FUNCTION_BLOCK CM_AX5000 EXTENDS CM_Base IMPLEMENTS I_AX5000
VAR_INPUT
	i_refAxis : REFERENCE TO Tc2_MC2.AXIS_REF;
	i_bIclkForward : BOOL := TRUE; //TRUE = interlocked
	i_bIclkBackward : BOOL := TRUE; //TRUE = interlocked
END_VAR

VAR
	fbPower : Tc2_MC2.MC_Power;
	fbReset : Tc2_MC2.MC_Reset;
	fbHome : Tc2_MC2.MC_Home;
	fbJog : Tc2_MC2.MC_Jog;
	fbMoveAbsolute : Tc2_MC2.MC_MoveAbsolute;
	fbMoveRelative : Tc2_MC2.MC_MoveRelative;
	fbStop : Tc2_MC2.MC_Stop;	

	// Inputs
	I_bDetReferenceSwitch AT %I* : BOOL; //Reference-/home switch
	I_bDetLimitSwitchPositive AT %I* : BOOL; //Limit switch positive-/CW- direction
	I_bDetLimitSwitchNegative AT %I* : BOOL; //Limit switch negative-/CCW- direction
	
	//Properties
	s_bStatus : BOOL;
	s_bDone : BOOL; 
	s_bBusy : BOOL; 
	s_bActive : BOOL; 
	s_bCommandAborted : BOOL; 
	s_bError : BOOL; 
	s_nErrorID : UDINT;
	
	// Requests
	{warning '#TODO: Chcek / update during develiping'}
	s_bReqStop : BOOL;
	s_bReqStartForward : BOOL;
	s_bReqStartBackward : BOOL;
	s_bReqReset : BOOL;
	
	// Commands
	s_bCmdEnable : BOOL;
	s_bCmdReset : BOOL;
	s_bCmdForward : BOOL;
	s_bCmdBackward : BOOL;
	s_bCmdReleaseBrake : BOOL;
		
	// States
	s_bStaReadyForOperation: BOOL;
	s_bStaDriveError: BOOL;
	s_bStaWarning : BOOL;
	
	
	
	s_sInterlockedReason : STRING; //External interlocked reason for clarifying reason
	
	// Setpoints
	s_fTargetSpeed : LREAL; // Target speed [mm/s]
	
	// Timers
	
	// Alarms
	s_fbAlarmHandlerDriveError : FB_AlarmHandler;
	s_fbAlarmHandlerStartMotorNotAllowed : FB_AlarmHandler;
	s_fbAlarmHandlerMotorForwardInterlocked : FB_AlarmHandler;
	s_fbAlarmHandlerMotorBackwardInterlocked : FB_AlarmHandler;
	
	s_errDriveError : BOOL;
	s_wrnStartMotorNotAllowed : BOOL;
	s_wrnMotorForwardInterlocked : BOOL;
	s_wrnMotorBackwardInterlocked : BOOL;
	
	//Hmi
	s_fbHmiBtnManualForward		: FB_HmiBtn;
	s_fbHmiBtnManualBackward	: FB_HmiBtn;
	s_fbHmiBtnManualStop		: FB_HmiBtn;
	s_fbHmiBtnManualReset		: FB_HmiBtn;
	
	s_fbHmiLedMotorStopped		: FB_HmiLed;
	s_fbHmiLedDriveError		: FB_HmiLed;
	
	//Sequence
	eSeqMOVITRAC_B_WithBrake : E_SeqMOVITRAC_B_WithBrake;
	seqTimer : TON;
	seqPreStep : E_SeqMOVITRAC_B_WithBrake;
	s_sActStep : STRING;
	
END_VAR


SUPER^();

METHOD PUBLIC m_MC_Home : BOOL
VAR_INPUT
	i_bExecute : BOOL;
	i_fPosition : REAL;
	i_eHomingMode : TC2_MC2.MC_HomingMode;
	i_eBufferMode : TC2_MC2.MC_BufferMode;
END_VAR

fbHome(
	Axis := i_refAxis,
	Execute := i_bExecute,
	Position := i_fPosition,
	HomingMode := i_eHomingMode,
	BufferMode := i_eBufferMode,
	Options := ,
	bCalibrationCam := I_bDetReferenceSwitch,
	Done => s_bDone,
	Busy => s_bBusy,
	Active => s_bActive,
	CommandAborted => s_bCommandAborted,
	Error => s_bError,
	ErrorID => s_nErrorID);
	
m_MC_Home := s_bDone;
END_METHOD

METHOD PUBLIC m_MC_Jog : BOOL
VAR_INPUT
	i_bExecute : BOOL;
	i_bJogForward : BOOL;
	i_bJogBackward : BOOL;
	i_eJogMode : TC2_MC2.E_JogMode;
	i_fPosition : LREAL; 
	i_fVelocity : LREAL; 
	i_fAcceleration : LREAL; 
	i_fDeceleration : LREAL; 
	i_fJerk : LREAL;
END_VAR

fbJog(
	Axis := i_refAxis,
	JogForward := i_bJogForward,
	JogBackwards := i_bJogBackward,
	Mode := i_eJogMode,
	Position := i_fPosition,
	Velocity := i_fVelocity,
	Acceleration := i_fAcceleration,
	Deceleration := i_fDeceleration,
	Jerk := i_fJerk,
	Done => s_bDone,
	Busy => s_bBusy,
	Active => s_bActive,
	CommandAborted => s_bCommandAborted,
	Error => s_bError,
	ErrorID => s_nErrorID);
	
m_MC_Home := s_bDone;
END_METHOD

METHOD PUBLIC m_MC_MoveAbsolute : BOOL
VAR_INPUT
	i_bExecute : BOOL;
	i_fPosition : LREAL; 
	i_fVelocity : LREAL; 
	i_fAcceleration : LREAL; 
	i_fDeceleration : LREAL; 
	i_fJerk : LREAL;
	i_eBufferMode : TC2_MC2.MC_BufferMode;
END_VAR

fbMoveAbsolute(
	Axis := i_refAxis,
	Execute := i_bExecute, 
	Position := i_fPosition,
	Velocity := i_fVelocity,
	Acceleration := i_fAcceleration,
	Deceleration := i_fDeceleration,
	Jerk := i_fJerk,
	BufferMode := i_eBufferMode,
	Options := ,
	Done => s_bDone,
	Busy => s_bBusy,
	Active => s_bActive,
	CommandAborted => s_bCommandAborted,
	Error => s_bError,
	ErrorID => s_nErrorID);
	
m_MC_Home := s_bDone;
END_METHOD

METHOD PUBLIC m_MC_MoveRelative : BOOL
VAR_INPUT
	i_bExecute : BOOL;
	i_fDistance : LREAL; 
	i_fVelocity : LREAL; 
	i_fAcceleration : LREAL; 
	i_fDeceleration : LREAL; 
	i_fJerk : LREAL;
	i_eBufferMode : TC2_MC2.MC_BufferMode;
END_VAR

fbMoveRelative(
	Axis := i_refAxis,
	Execute := i_bExecute,
	Distance := i_fDistance,
	Velocity := i_fVelocity,
	Acceleration := i_fAcceleration,
	Deceleration := i_fDeceleration,
	Jerk := i_fJerk,
	BufferMode := i_eBufferMode,
	Options := ,
	Done => s_bDone,
	Busy => s_bBusy,
	Active => s_bActive,
	CommandAborted => s_bCommandAborted,
	Error => s_bError,
	ErrorID => s_nErrorID);
	
m_MC_Home := s_bDone;
END_METHOD

METHOD PUBLIC m_MC_Power : BOOL
VAR_INPUT
	i_bEnable : BOOL;
	i_bEnablePositive : BOOL;
	i_bEnableNegative : BOOL;
	i_fOverride : LREAL;
	i_eBufferMode : TC2_MC2.MC_BufferMode;
END_VAR

fbPower(
	Axis := i_refAxis,
	Enable := i_bEnable,
	Enable_Positive := i_bEnablePositive,
	Enable_Negative := i_bEnableNegative,
	Override := i_fOverride,
	BufferMode := i_eBufferMode,
	Options := ,
	Status => s_bStatus,
	Busy => s_bBusy,
	Active => s_bActive,
	Error => s_bError,
	ErrorID => s_nErrorID);

m_MC_Home := s_bDone;
END_METHOD

METHOD PUBLIC m_MC_Reset : BOOL
VAR_INPUT
	i_bExecute : BOOL;
END_VAR

fbReset(
	Axis := i_refAxis,
	Execute := i_bExecute,
	Done => s_bDone,
	Busy => s_bBusy,
	Error => s_bError,
	ErrorID => s_nErrorID);

m_MC_Home := s_bDone;
END_METHOD

METHOD PUBLIC m_MC_Stop : BOOL
VAR_INPUT
	i_bExecute : BOOL;
	i_fDeceleration : LREAL;
	i_fJerk : LREAL;
END_VAR

fbStop(
	Axis := i_refAxis,
	Execute := i_bExecute,
	Deceleration := i_fDeceleration,
	Jerk := i_fJerk,
	Options := ,
	Done => s_bDone,
	Busy => s_bBusy,
	Active => s_bActive,
	CommandAborted => s_bCommandAborted,
	Error => s_bError,
	ErrorID => s_nErrorID);


m_MC_Home := s_bDone;
END_METHOD

PROPERTY PUBLIC p_bActive : BOOL
GET

p_bActive := s_bActive;
END_GET
END_PROPERTY

PROPERTY PUBLIC p_bBusy : BOOL
GET

p_bBusy := s_bBusy;
END_GET
END_PROPERTY

PROPERTY PUBLIC p_bCommandAborted : BOOL
GET

p_bCommandAborted := s_bCommandAborted
END_GET
END_PROPERTY

PROPERTY PUBLIC p_bDone : BOOL
GET

p_bDone := s_bDone
END_GET
END_PROPERTY

PROPERTY PUBLIC p_bError : BOOL
GET

p_bError := s_bError;
END_GET
END_PROPERTY

PROPERTY PUBLIC p_bHomed : BOOL
GET

p_bHomed := i_refAxis.Status.Homed;
END_GET
END_PROPERTY

PROPERTY PUBLIC p_bStandstill : BOOL
GET

p_bStandstill := i_refAxis.Status.StandStill;
END_GET
END_PROPERTY

PROPERTY PUBLIC p_fPosition : LREAL
GET

p_fPosition := i_refAxis.NcToPlc.ActPos;
END_GET
END_PROPERTY

PROPERTY PUBLIC p_fVelocity : LREAL
GET

p_fVelocity := i_refAxis.NcToPlc.ActVelo;
END_GET
END_PROPERTY

PROPERTY PUBLIC p_nErrorID : UDINT
GET

p_nErrorID := s_nErrorID;
END_GET
END_PROPERTY

END_FUNCTION_BLOCK

(* stored: Version 1.1.0.1, ProductVersion 3.1.4024.12
   POU CM_AX5000: Id {29dfdbae-f16d-497a-b262-2baea4701d77}, SpecialFunc None
   Folder Methods: Id {c7dc02dc-f2cb-44e5-89eb-2e4085b6a909}
   Folder Properties: Id {c3e008a7-9dfe-49e0-9cc5-18c79327535a}
   Method m_MC_Home: Id {953753d2-b56b-4416-8bfe-ffc202c2c66e}
   Method m_MC_Jog: Id {0b34f7cb-ad06-475a-9339-58c1a8e417e5}
   Method m_MC_MoveAbsolute: Id {0f6a7ef6-bbb9-453d-8d82-3eac920331b1}
   Method m_MC_MoveRelative: Id {e88d3f53-895e-4d90-93a1-00c818a65e17}
   Method m_MC_Power: Id {fd1fc676-b701-4a26-938f-ef477da725d4}
   Method m_MC_Reset: Id {78a60c41-19c8-4eb1-aa13-d3edbd9b9522}
   Method m_MC_Stop: Id {6c6294b9-0bc1-4c87-8f3e-41d07e1a757c}
   Property p_bActive: Id {fdebd466-4355-4961-86f7-17cb1e74e332}
   Get Get: Id {12554b68-dea8-473b-b98f-bf82edb9ad16}
   Property p_bBusy: Id {a6bb4214-9e42-46dd-a8f3-995e364772d0}
   Get Get: Id {7080bc48-c94e-419b-9e7d-df95694c753e}
   Property p_bCommandAborted: Id {32bd9d7d-f5a3-4f89-9a59-0294a826c560}
   Get Get: Id {a39acfdd-fde9-4118-9e65-bd86ad5a94af}
   Property p_bDone: Id {09a3960b-0e70-4e33-a3d6-ff5a57122d42}
   Get Get: Id {e656286c-fa2b-43ef-a794-1f2819d97be9}
   Property p_bError: Id {7759aec3-bd8b-4f0c-9913-656b2c70cf6a}
   Get Get: Id {67b5f8fe-c6e4-4145-9f0e-f9d36c480d63}
   Property p_bHomed: Id {29d86fc1-be45-4333-91ce-9bdc79739fba}
   Get Get: Id {3bff5f71-c84f-4863-9be2-8ae02d95a4db}
   Property p_bStandstill: Id {06fe4adf-3a6b-49c2-a8e8-c5de29d0c1af}
   Get Get: Id {e4db3dbb-9fbf-4ca7-ba91-332924a328ae}
   Property p_fPosition: Id {e5ef2cba-1955-4270-98db-4d1260096b27}
   Get Get: Id {440682b1-07c0-42c1-8793-ae28db2834f6}
   Property p_fVelocity: Id {e4d08808-aacd-469e-bccf-b788a2ac516e}
   Get Get: Id {a4e61425-56d9-43cd-b7a5-921c2a97d144}
   Property p_nErrorID: Id {063f18f8-6320-4761-b8fc-9920f5ec0c3a}
   Get Get: Id {fa545b5b-0766-4028-bde3-78e42d22c7e0} *)
